TYPE "UDT_HMI_Alarm_V2"
VERSION : 0.1
   STRUCT
      t : Struct
         x0 : Bool;
         x1 : Bool;
         x2 : Bool;
         x3 : Bool;
         x4 : Bool;
         x5 : Bool;
         x6 : Bool;
         x7 : Bool;
         x8 : Bool;
         x9 : Bool;
         x10 : Bool;
         x11 : Bool;
         x12 : Bool;
         x13 : Bool;
         x14 : Bool;
         x15 : Bool;
      END_STRUCT;
      iHmiSumAlm : Word;
   END_STRUCT;

END_TYPE

DATA_BLOCK "TiltingArms_Alm"
{ S7_Optimized_Access := 'FALSE' }
VERSION : 0.1
NON_RETAIN
   STRUCT
      tMotor : Array["STARTARRAY".."DNUMARM"] of Struct   // Motor allarms
         tEmergencyAlarm { ExternalWritable := 'False'} : Array["STARTARRAY".."DALARM"] of "UDT_HMI_Alarm_V2";
         tAlarm { ExternalWritable := 'False'} : Array["STARTARRAY".."DALARM"] of "UDT_HMI_Alarm_V2";
         tWarning { ExternalWritable := 'False'} : Array["STARTARRAY".."DALARM"] of "UDT_HMI_Alarm_V2";
      END_STRUCT;
      tEmergencyAlarm { S7_SetPoint := 'False'} : Array["STARTARRAY".."DALARM"] of "UDT_HMI_Alarm_V2";   // stop machine fault
      tAlarm { S7_SetPoint := 'False'} : Array["STARTARRAY".."DALARM"] of "UDT_HMI_Alarm_V2";   // stop next cycle faults
      tWarning { S7_SetPoint := 'False'} : Array["STARTARRAY".."DALARM"] of "UDT_HMI_Alarm_V2";   // Generic warning
   END_STRUCT;


BEGIN

END_DATA_BLOCK

DATA_BLOCK "TiltingArms_Hmi"
{ S7_Optimized_Access := 'FALSE' }
VERSION : 0.1
NON_RETAIN
   STRUCT
      tHMR : Struct   // {[Unit]|[Scada Unit]|[LowLimit]|[HigLimit]|[Acces]}
         tMotorSensor : Array["STARTARRAY".."DNUMARM"] of Struct   // Sensor status of motor
            xArmDown : Bool;
            xArmUp : Bool;
            xArmOk : Bool;
         END_STRUCT;
         dState : Int;   // State (1=no anomaly, 3= Run, 7=Anomaly) {x|x|x|x|O}
         dMotorState : Array["STARTARRAY".."DNUMARM"] of Int;   // State (1=no anomaly, 3= Run, 7=Anomaly) {x|x|x|x|O}
         tManCmd : Struct   // Manual commands Arm {x|x|x|x|O}
            xCmdLift : Array["STARTARRAY".."DNUMARM"] of Bool;   // Manual Command Lift Arm {x|x|x|x|O}
            xCmdDescent : Array["STARTARRAY".."DNUMARM"] of Bool;   // Manual Command Descent Arm {x|x|x|x|O}
            xCmdLiftAll : Bool;
            xCmdDescentAll : Bool;
         END_STRUCT;
      END_STRUCT;
      tHMW : Struct   // {[Unit]|[Scada Unit]|[LowLimit]|[HigLimit]|[Acces]}
         tManCmd : Struct   // Manual commands Arm {x|x|x|x|O}
            xCmdLift : Array["STARTARRAY".."DNUMARM"] of Bool;   // Manual Command Lift Arm {x|x|x|x|O}
            xCmdDescent : Array["STARTARRAY".."DNUMARM"] of Bool;   // Manual Command Descent Arm {x|x|x|x|O}
            xCmdLiftAll : Bool;
            xCmdDescentAll : Bool;
         END_STRUCT;
      END_STRUCT;
   END_STRUCT;


BEGIN

END_DATA_BLOCK

